# EPICS autosave request: hexapodApp/Db/asyn_motor_positions.req
# FILE... motor_positions.req
$(P)$(M).DVAL
